Staubli VAL3: Control_Action.pgx

public program Control_Action(num& x_nAction[] (dimensions=3), num x_nIndex, string& x_sIoName[], bool& x_bDigtal[])
  local string l_sItem[2]
  local num l_nNum
  local num l_nKey
  local num l_nData[24]
  local num l_nSelectIndex
  local bool l_bRes
  local num l_nBuff
begin
  //为LasMAN3.7 Action配置


  for l_nNum=0 to 11
    l_nData[l_nNum*2+0]=x_nAction[x_nIndex,l_nNum,0]
    l_nData[l_nNum*2+1]=x_nAction[x_nIndex,l_nNum,1]
  endFor
  l_sItem[0]="关"
  l_sItem[1]="开"

  resize(sBuff,1,24)


  call Control_BottomS("置空,清空,延时,插入,删除,,取消,确定")
  call Control_PanelXY(4,0,20,10)
  call Control_Panel("动作值")
  for l_nNum=0 to 11


    sBuff[l_nNum*2+0]=toString("",l_nNum+1)+"名称:"+x_sIoName[l_nData[l_nNum*2+0]]
    if x_bDigtal[l_nData[l_nNum*2]]
      sBuff[l_nNum*2+1]="值 : "+ l_sItem[sel(l_nData[l_nNum*2+1]==0,0,1)]
    else
      sBuff[l_nNum*2+1]="值 : "+toString(".1",l_nData[l_nNum*2+1])
    endIf

  endFor
  call Control_List(sBuff,l_nSelectIndex)


  //**********************************
  //按键响应
  while true
    l_nKey=getKey()

    switch l_nKey
      //向上
      case 261
        l_nSelectIndex=max(0,l_nSelectIndex-1)
      break

      //向下
      case 266
        l_nSelectIndex=min(l_nSelectIndex+1,23)
      break

      //编辑
      case 270
        if l_nSelectIndex%2==1
          if ! x_bDigtal[l_nData[l_nSelectIndex-1]]
            call Float_Edit(l_nData[l_nSelectIndex],nPanelLTopX+6,l_nSelectIndex+nPanelLTopY+1)
          else
            l_nData[l_nSelectIndex]=sel(l_nData[l_nSelectIndex]==1,1,0)
            call Sel_Edit(l_nData[l_nSelectIndex],nPanelLTopX+6,l_nSelectIndex+nPanelLTopY+1,l_sItem)
            l_nData[l_nSelectIndex]=sel(l_nData[l_nSelectIndex]==1,1,0)
          endIf

        else
          call Sel_Edit(l_nData[l_nSelectIndex],nPanelLTopX+7,l_nSelectIndex+nPanelLTopY+1,x_sIoName)
        endIf

      break

      case 271
        call Control_YesNO("确定设置为无IO信号吗?",l_bRes)
        if l_bRes

          l_nData[sel(l_nSelectIndex%2==0,l_nSelectIndex,l_nSelectIndex-1)]=0

        endIf

      break


      //全部置空
      case 272
        call Control_YesNO("确定全部清空吗?",l_bRes)
        if l_bRes
          for l_nNum=0 to 23
            l_nData[l_nNum]=0
          endFor


        endIf
      break


      case 273
        call Control_YesNO("确定要设置为延时吗?",l_bRes)
        if l_bRes
          l_nData[sel(l_nSelectIndex%2==0,l_nSelectIndex,l_nSelectIndex-1)]=165

        endIf
      break

      //插入
      case 274
        call Control_YesNO("确定要插入吗?",l_bRes)
        l_nBuff=roundDown(l_nSelectIndex/2)
        if l_bRes
          for l_nNum=23 to l_nBuff*2+2  step -1
            l_nData[l_nNum]=l_nData[l_nNum-2]
          endFor
          l_nData[l_nBuff*2]=l_nData[l_nBuff*2+1]=0

        endIf
      break


      //删除
      case 275
        call Control_YesNO("确定要删除吗?",l_bRes)
        l_nBuff=roundDown(l_nSelectIndex/2)
        if l_bRes
          for l_nNum=l_nBuff*2 to 21
            l_nData[l_nNum]=l_nData[l_nNum+2]
          endFor
          l_nData[23]=l_nData[22]=0

        endIf
      break





      //退出
      case 277
        cls()
        return

      break



      //取消
      case 278
        for l_nNum=0 to 11
          x_nAction[x_nIndex,l_nNum,0]= l_nData[l_nNum*2+0]
          x_nAction[x_nIndex,l_nNum,1]=l_nData[l_nNum*2+1]
        endFor
        return
      break

    endSwitch

    if l_nKey!=-1

      for l_nNum=0 to 11
        sBuff[l_nNum*2+0]=toString("",l_nNum+1)+"名称:"+x_sIoName[l_nData[l_nNum*2+0]]
        if x_bDigtal[l_nData[l_nNum*2]]
          sBuff[l_nNum*2+1]="值 : "+ l_sItem[sel(l_nData[l_nNum*2+1]==0,0,1)]
        else
          sBuff[l_nNum*2+1]="值 : "+toString(".2",l_nData[l_nNum*2+1])
        endIf

      endFor

      call Control_PanelXY(4,0,20,10)
      call Control_Panel("动作值")
      call Control_List(sBuff,l_nSelectIndex)
      call Control_BottomS("置空,清空,延时,插入,删除,,取消,确定")
    endIf


  endWhile





end
